SUBAPPLICATION Uebung_034a1_Q1 (* Numeric Value Input auf PWM Ausgang *)
  (* Standard: 61499-2; Description: Copyright (c) 2023 Meisterschulen am Ostbahnhof This program and the accompanying materials are made available under the terms of the Eclipse Public License 2.0 which is available at https://www.eclipse.org/legal/epl-2.0/ SPDX-License-Identifier: EPL-2.0 *)
  (* Version 1.0, 2023-10-23, Franz Höpfinger, Meisterschulen am Ostbahnhof *)
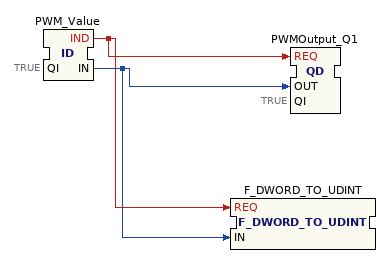
  (* ACHTUNG !! IND erscheint erst, wenn man die Numeric Value mit OK Bestätigt. nicht bei Button Druck. *)
  FBS
    F_DWORD_TO_UDINT : F_DWORD_TO_UDINT;
    PWMOutput_Q1 : QD(QI := TRUE);
    PWM_Value : ID(QI := TRUE);
  END_FBS
  EVENT_CONNECTIONS
    PWM_Value.IND TO PWMOutput_Q1.REQ;
    PWM_Value.IND TO F_DWORD_TO_UDINT.REQ;
  END_CONNECTIONS
  DATA_CONNECTIONS
    PWM_Value.IN TO F_DWORD_TO_UDINT.IN;
    PWM_Value.IN TO PWMOutput_Q1.OUT;
  END_CONNECTIONS
END_SUBAPPLICATION
